(* CODESYS project systemdk.library
   Company: Beckhoff - DK
   DefaultNamespace: Tc3_SystemDK
   Title: Tc3_SystemDK
   Placeholder: Tc3_SystemDK
   Author: HCP
   Version: 3.3.1.5

Project tree, tasks and I/O mapping:
  libraries: Tc2_EtherCAT, * (Beckhoff Automation GmbH); Tc2_IoFunctions, * (Beckhoff Automation GmbH); Tc2_Standard, * (Beckhoff Automation GmbH); Tc2_SUPS, * (Beckhoff Automation GmbH); Tc2_System, * (Beckhoff Automation GmbH); Tc2_Utilities, * (Beckhoff Automation GmbH); Tc3_Interfaces, * (Beckhoff Automation GmbH); Tc3_Module, * (Beckhoff Automation GmbH)
  BASIC/
    POUs/
      FBs/
        DUTs/
          data type ST_Basic
          data type ST_Basic_Status
        GVLs/
          global variables GVL_Basic
        ITFs/
          interface I_Basic: M_nError, M_nReset, P_bAuto, P_bError, P_bManual, P_bReady, P_bReset, P_nErrorID
        function block FB_Basic [ST]: M_nError, M_nReset, P_bAuto, P_bError, P_bManual, P_bReady, P_bReset, P_nErrorID
  SYSTEM/
    POUs/
      FBs/
        DUTs/
          data type ST_EtherCATStatusDK
          data type ST_NovRamDK
          data type ST_SystemDK
          data type ST_WritePersistentDataDK
        ITFs/
          interface I_EtherCATStatusDK: M_nEnable, P_bWireBroke, P_nCfgSlaveCount, P_nDevState, P_nSlaveCount
          interface I_NovRamDK: M_nEnable
          interface I_SystemDK: M_nCerHost, M_nEnable, P_bIs_ARM, P_bIs_CE_Device, P_bIs_x64, P_bIs_x86, P_nAdsPort, P_nCycleTime, P_stDeviceIdentificationEx
          interface I_WritePersistentDataDK: M_n1_Second_UPS, M_nEnable, M_nWrite, P_bBusy, P_bPowerFailDetect, P_eSUPS_Mode, P_nWriteCNT
        function block FB_EtherCATStatusDK [ST]: M_nEnable, P_bWireBroke, P_nCfgSlaveCount, P_nDevState, P_nSlaveCount
        function block FB_NovRamDK [ST]: M_nEnable, M_nRead, M_nWrite
        function block FB_SystemDK [ST]: M_nCerHost, M_nEnable, P_bIs_ARM, P_bIs_CE_Device, P_bIs_x64, P_bIs_x86, P_nAdsPort, P_nCycleTime, P_stDeviceIdentificationEx
        function block FB_WritePersistentDataDK [ST]: M_n1_Second_UPS, M_nEnable, M_nWrite, P_bBusy, P_bPowerFailDetect, P_eSUPS_Mode, P_nWriteCNT
  Version/
    global variables Global_Version
*)

// BASIC/POUs/FBs/DUTs/ST_Basic
TYPE ST_Basic :
STRUCT
	bAuto: BOOL;
	bManual: BOOL;
	bReady: BOOL;
	bReset: BOOL;
	bError: BOOL;
	nErrorID: UDINT;
	nStatus: UDINT;	
	arr_nStatus: ARRAY[1..20] OF UDINT;
END_STRUCT
END_TYPE

// BASIC/POUs/FBs/DUTs/ST_Basic_Status
TYPE ST_Basic_Status :
STRUCT
	nError: UDINT;
	nReset:UDINT;
END_STRUCT
END_TYPE

// SYSTEM/POUs/FBs/DUTs/ST_EtherCATStatusDK
TYPE ST_EtherCATStatusDK EXTENDS ST_Basic :
STRUCT
	nDevState: UINT;
	nSlaveCount: UINT;
	nCfgSlaveCount: UINT;
	
	bWireBroke: BOOL;
END_STRUCT
END_TYPE

// SYSTEM/POUs/FBs/DUTs/ST_NovRamDK
TYPE ST_NovRamDK EXTENDS ST_Basic :
STRUCT
	bEnable: BOOL;
END_STRUCT
END_TYPE

// SYSTEM/POUs/FBs/DUTs/ST_SystemDK
TYPE ST_SystemDK EXTENDS ST_Basic :
STRUCT
	bIs_CE_Device: BOOL;			// Is a CE Device
	bIs_ARM: BOOL;					// Is ARM runtime
	bIs_x86: BOOL;					// Is x86 runtime
	bIs_x64: BOOL;					// Is x64 runtime
	nAdsPort: UINT;					// Plc port nr
	nCycleTime: UDINT;				// Plc cycle time in 100nS
	bCerHost_Enable: BOOL;			// Enable CerHost
	bCerHost_Disable: BOOL;			// Disable CerHost
	stDeviceIdentificationEx: Tc2_Utilities.ST_DeviceIdentificationEx;
END_STRUCT
END_TYPE

// SYSTEM/POUs/FBs/DUTs/ST_WritePersistentDataDK
TYPE ST_WritePersistentDataDK EXTENDS ST_Basic :
STRUCT
	bWrite: BOOL;
	bBusy: BOOL;
	bPowerFailDetect: BOOL;
	nWriteCNT: UDINT;
END_STRUCT
END_TYPE

// BASIC/POUs/FBs/GVLs/GVL_Basic
VAR_GLOBAL CONSTANT
	cIDLE: UDINT:= 0;						//	0 = idle
	cCOUPLED: UDINT:= 1;					//	1 = coupled
	cSTARTING: UDINT:= 2;					//	2 = starting
	cRUNNING: UDINT:= 3;					//	3 = running
	cABORTED: UDINT:= 4;					//	4 = aborted
	cNO_HARDWARE_CONNECTED: UDINT:= 5;		// 	5 = no hardware connected
	
	cPOINTER_OR_INDEX_ERROR: UDINT:= 7;		//	7 = pointer or index error
	cMAPPING_ERROR: UDINT:= 8;				//	8 = mapping error
	cPARAMETER_ERROR: UDINT:= 9;			//	9 = parameter error
	cCOMPLETE: UDINT:= 10;					//	10 = complete
END_VAR

// Version/Global_Version
// This function has been automatically generated from the project information.
VAR_GLOBAL CONSTANT
	{attribute 'const_non_replaced'}
	{attribute 'linkalways'}
	stLibVersion_Tc3_SystemDK : ST_LibVersion := (iMajor := 3, iMinor := 3, iBuild := 1, iRevision := 5, sVersion := '3.3.1.5');
END_VAR

// BASIC/POUs/FBs/ITFs/I_Basic
INTERFACE I_Basic

//	The result of the method is an unsigned double integer
//	0 = idle 
//	1 = coupled
//	2 = starting
//	3 = running
//	4 = aborted
// 	5 = no hardware connected
//	7 = pointer or index error
//	8 = mapping error
//	9 = parameter error
//	10 = complete
//	Any other number = ErrorID
METHOD PUBLIC M_nError : UDINT
VAR_INPUT
	nErrorID: UDINT;
END_VAR
END_METHOD

//	The result of the method is an unsigned double integer
//	0 = idle 
//	1 = coupled
//	2 = starting
//	3 = running
//	4 = aborted
// 	5 = no hardware connected
//	7 = pointer or index error
//	8 = mapping error
//	9 = parameter error
//	10 = complete
//	Any other number = ErrorID
METHOD PUBLIC M_nReset : UDINT
VAR_INPUT
	bExecute: BOOL;
END_VAR
END_METHOD

PROPERTY PUBLIC P_bAuto : BOOL
GET
END_GET
SET
END_SET
END_PROPERTY

PROPERTY PUBLIC P_bError : BOOL
GET
END_GET
END_PROPERTY

PROPERTY PUBLIC P_bManual : BOOL
GET
END_GET
SET
END_SET
END_PROPERTY

PROPERTY PUBLIC P_bReady : BOOL
GET
END_GET
SET
END_SET
END_PROPERTY

PROPERTY PUBLIC P_bReset : BOOL
GET
END_GET
END_PROPERTY

PROPERTY PUBLIC P_nErrorID : UDINT
GET
END_GET
END_PROPERTY

END_INTERFACE

// BASIC/POUs/FBs/FB_Basic
//------------------------------------------------------------------------------------------
//                                                                                        	
//***************************** Beckhoff TwinCAT Examples **********************************
//                                                                                        	
//************************************* WARNING ********************************************
// This program is only an example. If it is used as a control program in any real        	
// application, Beckhoff is not responsible for any malfunction, loss or damage           	
// which could arise by using this program!                                               	
//                                                                                        	
//*************************************  Program Info. *************************************
//                                                                                        	
// PLC program name:       FB_Basic (FB)               	                           	
// Hardware platform:      TwinCat v3.1.4012				                          	
// Modified by:            Hans Chr. Pallesen 			                                  	
//                                                                                        	
// ======================================================================================== 
//         Version       Date                        Remarks                              	
// ======================================================================================== 
//         1.0           17 feb 2013                 First release of this example        	
//         1.1           05 aug 2013                 Next release of this example        	
//         1.2           10 dec 2013                 Next release of this example        	
//         1.3           12 mar 2014                 Next release of this example        	
//         1.4           28 mar 2014                 Next release of this example        	
//         1.5           02 jun 2014                 Next release of this example        	
// ======================================================================================== 
//                                                                                        	
//******************************* Aims OF this PLC PROGRAM *********************************
//                                                                                        	
// Basic FB  						 			                               	
//																	                      	
//                                                                                        	
//----------------------------------------------------------------------------------------- 
FUNCTION_BLOCK FB_Basic IMPLEMENTS I_Basic
VAR
	_iIdx: INT;		// Temporary variabel - Index pointer
	
//*************************
// Property variables
//*************************
	_bReset: BOOL;
	_bAuto: BOOL := TRUE;
	_bManual: BOOL;
	_bError: BOOL;
	_nErrorID: UDINT;
	_bReady: BOOL;
	
//*************************
// Methods variable
//*************************
	FB_Basic_M_nReset_nScanCNT: UINT;
	FB_Basic_M_nReset_fbR_TRIG: Tc2_Standard.R_TRIG;
END_VAR

//	The result of the method is an unsigned double integer
//	0 = idle 
//	1 = coupled
//	2 = starting
//	3 = running
//	4 = aborted
// 	5 = no hardware connected
//	7 = pointer or index error
//	8 = mapping error
//	9 = parameter error
//	10 = complete
//	Any other number = ErrorID
METHOD PUBLIC M_nError : UDINT
VAR_INPUT
	nErrorID: UDINT;
END_VAR
//**********************************
// Update error
//**********************************
IF NOT _bError THEN
	_nErrorID:= nErrorID;
	_bError:= TRUE;
END_IF

M_nError:= cCOMPLETE;
END_METHOD

//	The result of the method is an unsigned double integer
//	0 = idle 
//	1 = coupled
//	2 = starting
//	3 = running
//	4 = aborted
// 	5 = no hardware connected
//	7 = pointer or index error
//	8 = mapping error
//	9 = parameter error
//	10 = complete
//	Any other number = ErrorID
METHOD PUBLIC M_nReset : UDINT
VAR_INPUT
	bExecute: BOOL;
END_VAR
//**********************************
// Wait for execute
//**********************************
FB_Basic_M_nReset_fbR_TRIG(CLK:= bExecute);
IF FB_Basic_M_nReset_fbR_TRIG.Q THEN
	FB_Basic_M_nReset_nScanCNT:= 4;	
	_bReset:= TRUE;
ELSE
	// Delay
	IF FB_Basic_M_nReset_nScanCNT = 0 THEN
		_bReset:= FALSE;
	ELSE
		IF FB_Basic_M_nReset_nScanCNT <= 2 THEN
			_bError:= FALSE;
			_nErrorID:= 16#00;
		END_IF	
	END_IF

	// Scan counter
	IF FB_Basic_M_nReset_nScanCNT > 0 THEN
		FB_Basic_M_nReset_nScanCNT:= FB_Basic_M_nReset_nScanCNT -1;
	ELSE	
		FB_Basic_M_nReset_nScanCNT:= 0;
	END_IF

	// Return method state
	IF bExecute THEN
		IF FB_Basic_M_nReset_nScanCNT = 0 THEN
			M_nReset:= cCOMPLETE;
		ELSE
			M_nReset:= cRUNNING;
		END_IF
	ELSE	
		M_nReset:= cIDLE;
	END_IF	
END_IF
END_METHOD

PROPERTY PUBLIC P_bAuto : BOOL
GET
P_bAuto:= _bAuto;
END_GET
SET
_bAuto:= P_bAuto;
END_SET
END_PROPERTY

PROPERTY PUBLIC P_bError : BOOL
GET
P_bError:= _bError;
END_GET
END_PROPERTY

PROPERTY PUBLIC P_bManual : BOOL
GET
P_bManual:= _bManual;
END_GET
SET
_bManual:= P_bManual;
END_SET
END_PROPERTY

PROPERTY PUBLIC P_bReady : BOOL
GET
P_bReady:= _bReady;
END_GET
SET
PUBLIC 
VAR
END_VAR
_bReady:= P_bReady;
END_SET
END_PROPERTY

PROPERTY PUBLIC P_bReset : BOOL
GET
P_bReset:= _bReset;
END_GET
END_PROPERTY

PROPERTY PUBLIC P_nErrorID : UDINT
GET
P_nErrorID:= _nErrorID;
END_GET
END_PROPERTY

END_FUNCTION_BLOCK

// SYSTEM/POUs/FBs/ITFs/I_EtherCATStatusDK
INTERFACE I_EtherCATStatusDK EXTENDS I_Basic

//	The result of the method is an unsigned double integer
//	0 = idle 
//	1 = coupled
//	2 = starting
//	3 = running
//	4 = aborted
// 	5 = no hardware connected
//	7 = pointer or index error
//	8 = mapping error
//	9 = parameter error
//	10 = complete
//	Any other number = ErrorID
METHOD PUBLIC M_nEnable : UDINT
VAR_INPUT
	bExecute: BOOL;
END_VAR
END_METHOD

PROPERTY PUBLIC P_bWireBroke : BOOL
GET
END_GET
END_PROPERTY

PROPERTY PUBLIC P_nCfgSlaveCount : UINT
GET
END_GET
END_PROPERTY

PROPERTY PUBLIC P_nDevState : UINT
GET
END_GET
END_PROPERTY

PROPERTY PUBLIC P_nSlaveCount : UINT
GET
END_GET
END_PROPERTY

END_INTERFACE

// SYSTEM/POUs/FBs/ITFs/I_NovRamDK
INTERFACE I_NovRamDK EXTENDS I_Basic

//	The result of the method is an unsigned double integer
//	0 = idle 
//	1 = coupled
//	2 = starting
//	3 = running
//	4 = aborted
// 	5 = no hardware connected
//	7 = pointer or index error
//	8 = mapping error
//	9 = parameter error
//	10 = complete
//	Any other number = ErrorID
METHOD M_nEnable : UDINT
VAR_INPUT
	bExecute: BOOL;
	nDevId: UINT;
	nMB_Offset: UINT;
	nMB_Size: UINT;
END_VAR
END_METHOD

END_INTERFACE

// SYSTEM/POUs/FBs/ITFs/I_SystemDK
INTERFACE I_SystemDK EXTENDS I_Basic

//	The result of the method is an unsigned double integer
//	0 = idle 
//	1 = coupled
//	2 = starting
//	3 = running
//	4 = aborted
// 	5 = no hardware connected
//	7 = pointer or index error
//	8 = mapping error
//	9 = parameter error
//	10 = complete
//	Any other number = ErrorID
METHOD PUBLIC M_nCerHost : UDINT
VAR_INPUT
	bEnable: BOOL;
	bDisable: BOOL;
END_VAR
END_METHOD

//	The result of the method is an unsigned double integer
//	0 = idle 
//	1 = coupled
//	2 = starting
//	3 = running
//	4 = aborted
// 	5 = no hardware connected
//	7 = pointer or index error
//	8 = mapping error
//	9 = parameter error
//	10 = complete
//	Any other number = ErrorID
METHOD PUBLIC M_nEnable : UDINT
VAR_INPUT
END_VAR
END_METHOD

PROPERTY PUBLIC P_bIs_ARM : BOOL
GET
END_GET
END_PROPERTY

PROPERTY PUBLIC P_bIs_CE_Device : BOOL
GET
END_GET
END_PROPERTY

PROPERTY PUBLIC P_bIs_x64 : BOOL
GET
END_GET
END_PROPERTY

PROPERTY PUBLIC P_bIs_x86 : BOOL
GET
END_GET
END_PROPERTY

PROPERTY PUBLIC P_nAdsPort : UINT
GET
END_GET
END_PROPERTY

PROPERTY PUBLIC P_nCycleTime : UDINT
GET
END_GET
END_PROPERTY

PROPERTY PUBLIC P_stDeviceIdentificationEx : Tc2_Utilities.ST_DeviceIdentificationEx
GET
END_GET
END_PROPERTY

END_INTERFACE

// SYSTEM/POUs/FBs/ITFs/I_WritePersistentDataDK
INTERFACE I_WritePersistentDataDK EXTENDS I_Basic

//	The result of the method is an unsigned double integer
//	0 = idle 
//	1 = coupled
//	2 = starting
//	3 = running
//	4 = aborted
// 	5 = no hardware connected
//	7 = pointer or index error
//	8 = mapping error
//	9 = parameter error
//	10 = complete
//	Any other number = ErrorID
METHOD PUBLIC M_n1_Second_UPS : UDINT
VAR_INPUT
	bExecute: BOOL;
END_VAR
END_METHOD

//	The result of the method is an unsigned double integer
//	0 = idle 
//	1 = coupled
//	2 = starting
//	3 = running
//	4 = aborted
// 	5 = no hardware connected
//	7 = pointer or index error
//	8 = mapping error
//	9 = parameter error
//	10 = complete
//	Any other number = ErrorID
METHOD M_nEnable : UDINT
VAR_INPUT
	bExecute: BOOL;
	tLogTimePuls: TIME;
END_VAR
END_METHOD

//	The result of the method is an unsigned double integer
//	0 = idle 
//	1 = coupled
//	2 = starting
//	3 = running
//	4 = aborted
// 	5 = no hardware connected
//	7 = pointer or index error
//	8 = mapping error
//	9 = parameter error
//	10 = complete
//	Any other number = ErrorID
METHOD M_nWrite : UDINT
VAR_INPUT
	bExecute: BOOL;
END_VAR
END_METHOD

PROPERTY PUBLIC P_bBusy : BOOL
GET
END_GET
END_PROPERTY

PROPERTY PUBLIC P_bPowerFailDetect : BOOL
GET
END_GET
END_PROPERTY

PROPERTY PUBLIC P_eSUPS_Mode : Tc2_SUPS.E_S_UPS_Mode
SET
END_SET
END_PROPERTY

PROPERTY PUBLIC P_nWriteCNT : UDINT
GET
END_GET
END_PROPERTY

END_INTERFACE

// SYSTEM/POUs/FBs/FB_EtherCATStatusDK
//------------------------------------------------------------------------------------------
//                                                                                        	
//***************************** Beckhoff TwinCAT Examples **********************************
//                                                                                        	
//************************************* WARNING ********************************************
// This program is only an example. If it is used as a control program in any real        	
// application, Beckhoff is not responsible for any malfunction, loss or damage           	
// which could arise by using this program!                                               	
//                                                                                        	
//*************************************  Program Info. *************************************
//                                                                                        	
// PLC program name:       FB_EtherCAT_Ok (FB)                                          	
// Hardware platform:      TwinCat v3.1.4014				                          	
// Modified by:            Hans Chr. Pallesen 			                                  	
//                                                                                        	
// ======================================================================================== 
//         Version       Date                        Remarks                              	
// ======================================================================================== 
//         1.0           12 feb 2014                 First release of this example        	
// ======================================================================================== 
//                                                                                        	
//******************************* Aims OF this PLC PROGRAM *********************************
//                                                                                        	
// Check EtherCAT state				 			                                      	
//																	                      	
//                                                                                        	
//----------------------------------------------------------------------------------------- 
FUNCTION_BLOCK FB_EtherCATStatusDK EXTENDS FB_Basic IMPLEMENTS I_EtherCATStatusDK
VAR
//**************************
// Static variables
//**************************
	AI_DevState AT %I*: UINT;
	AI_SlaveCount AT %I*: UINT;
	AI_CfgSlaveCount AT %I*: UINT;
//**************************
// Property variables
//**************************
	_bWireBroke: BOOL;
	
//**********************************
// Methods variable
//**********************************
	FB_EtherCATStatus_M_nEnable_fbDelay_TON: Tc2_Standard.TON;
END_VAR

//	The result of the method is an unsigned double integer
//	0 = idle 
//	1 = coupled
//	2 = starting
//	3 = running
//	4 = aborted
// 	5 = no hardware connected
//	7 = pointer or index error
//	8 = mapping error
//	9 = parameter error
//	10 = complete
//	Any other number = ErrorID
METHOD PUBLIC M_nEnable : UDINT
VAR_INPUT
	bExecute: BOOL;
END_VAR
// EtherCAT not configered
IF AI_SlaveCount = 0 AND AI_CfgSlaveCount = 0 THEN
	_bReady:= FALSE;
	_bWireBroke:= FALSE;
	M_nEnable:= cNO_HARDWARE_CONNECTED; 
ELSE
	// EtherCAT used
	IF bExecute THEN
		
		// Update Wire broke
		IF (AI_SlaveCount = 0 OR AI_SlaveCount <> AI_CfgSlaveCount) THEN
			M_nError(nErrorID:= 0);	
			_bWireBroke:= TRUE;
		ELSE
			_bWireBroke:= FALSE;
		END_IF
		
		// Update DevState
		IF AI_DevState <> 0 THEN
			M_nError(nErrorID:= 0);	
		END_IF
		
		// Method return value
		FB_EtherCATStatus_M_nEnable_fbDelay_TON(IN:= NOT _bWireBroke AND (AI_DevState = 0), PT:= T#100MS);
		_bReady:= FB_EtherCATStatus_M_nEnable_fbDelay_TON.Q;
		
		// Check for hardware
		IF AI_SlaveCount = 0 THEN
			M_nEnable:= cNO_HARDWARE_CONNECTED;
		ELSE
			IF _bReady THEN
				M_nEnable:= cCOMPLETE;
			ELSE
				M_nEnable:= cIDLE;
			END_IF
		END_IF
		
	ELSE
		FB_EtherCATStatus_M_nEnable_fbDelay_TON(IN:= FALSE);
		_bReady:= FALSE;
		_bWireBroke:= FALSE;
		M_nEnable:= cIDLE; 
	END_IF	

END_IF
END_METHOD

PROPERTY PUBLIC P_bWireBroke : BOOL
GET
P_bWireBroke:= _bWireBroke;
END_GET
END_PROPERTY

PROPERTY PUBLIC P_nCfgSlaveCount : UINT
GET
P_nCfgSlaveCount:= AI_CfgSlaveCount;
END_GET
END_PROPERTY

PROPERTY PUBLIC P_nDevState : UINT
GET
P_nDevState:= AI_DevState;
END_GET
END_PROPERTY

PROPERTY PUBLIC P_nSlaveCount : UINT
GET
P_nSlaveCount:= AI_SlaveCount;
END_GET
END_PROPERTY

END_FUNCTION_BLOCK

// SYSTEM/POUs/FBs/FB_NovRamDK
//------------------------------------------------------------------------------------------
//                                                                                        	
//***************************** Beckhoff TwinCAT Examples **********************************
//                                                                                        	
//************************************* WARNING ********************************************
// This program is only an example. If it is used as a control program in any real        	
// application, Beckhoff is not responsible for any malfunction, loss or damage           	
// which could arise by using this program!                                               	
//                                                                                        	
//*************************************  Program Info. *************************************
//                                                                                        	
// PLC program name:       FB_NovRamDK (FB)               	                           	
// Hardware platform:      TwinCat v3.1.4012				                          	
// Modified by:            Hans Chr. Pallesen 			                                  	
//                                                                                        	
// ======================================================================================== 
//         Version       Date                        Remarks                              	
// ======================================================================================== 
//         1.0           27 nov 2013                 First release of this example        	
// ======================================================================================== 
//                                                                                        	
//******************************* Aims OF this PLC PROGRAM *********************************
//                                                                                        	
//	Read/Write to NovRam																	                      	
//                                                                                        	
//----------------------------------------------------------------------------------------- 
FUNCTION_BLOCK FB_NovRamDK EXTENDS FB_Basic IMPLEMENTS I_NovRamDK
VAR
//**********************************
// Static variables
//**********************************
	_bEnable: BOOL;
	_nDevId: UINT;
	_nMB_Offset: UINT;
	_nMB_Size: UINT;
//**********************************
// Methods variable
//**********************************
	FB_NovRamDK_M_nEnable_nMBSrc AT %MB0: BYTE;
	FB_NovRamDK_M_nEnable_nBank: BYTE;
	FB_NovRamDK_M_nEnable_nCalcSize: UINT;
	FB_NovRamDK_M_nEnable_iState: UINT;
	FB_NovRamDK_M_nEnable_fbExecute_R_TRIG: Tc2_Standard.R_TRIG;
	FB_NovRamDK_M_nEnable_fbExecute_F_TRIG: Tc2_Standard.F_TRIG;
	FB_NovRamDK_M_nEnable_fbGetDPRAMInfo: Tc2_IoFunctions.FB_GetDPRAMInfo;
	FB_NovRamDK_M_nEnable_stNovRamAddrInfo: Tc2_IoFunctions.ST_NovRamAddrInfo;
	FB_NovRamDK_M_nEnable_nArrStatus: ARRAY[1..5] OF UDINT;

	FB_NovRamDK_M_nRead_fbNovRamReadWriteEx: FB_NovRamReadWriteEx;
	FB_NovRamDK_M_nRead_iState: UINT;
	FB_NovRamDK_M_nRead_nBank: BYTE;

	FB_NovRamDK_M_nWrite_fbNovRamReadWriteEx: FB_NovRamReadWriteEx;
	FB_NovRamDK_M_nWrite_bReady: BOOL;
	FB_NovRamDK_M_nWrite_iState: UINT;
	FB_NovRamDK_M_nWrite_nBank: BYTE;
	FB_NovRamDK_M_nWrite_pByte: POINTER TO BYTE;
	FB_NovRamDK_M_nWrite_pCard: POINTER TO BYTE;
END_VAR

//	The result of the method is an unsigned double integer
//	0 = idle 
//	1 = coupled
//	2 = starting
//	3 = running
//	4 = aborted
// 	5 = no hardware connected
//	7 = pointer or index error
//	8 = mapping error
//	9 = parameter error
//	10 = complete
//	Any other number = ErrorID
METHOD PUBLIC M_nEnable : UDINT
VAR_INPUT
	bExecute: BOOL;
	nDevId: UINT;
	nMB_Offset: UINT;
	nMB_Size: UINT;
END_VAR
//**********************************
// Local variable
//**********************************
THIS^._bEnable:= bExecute;
THIS^._nDevId:= nDevId;
THIS^._nMB_Offset:= nMB_Offset;
THIS^._nMB_Size:= nMB_Size;

//**********************************
// Reset
//**********************************
IF _bReset THEN
	IF _bError THEN
		FB_NovRamDK_M_nEnable_iState:= 000;
	END_IF
	M_nReset(bExecute:= _bReset);
END_IF

//**********************************
// Wait for execute
//**********************************
FB_NovRamDK_M_nEnable_fbExecute_R_TRIG(CLK:= bExecute);
FB_NovRamDK_M_nEnable_fbExecute_F_TRIG(CLK:= bExecute);
IF FB_NovRamDK_M_nEnable_fbExecute_R_TRIG.Q OR FB_NovRamDK_M_nEnable_fbExecute_F_TRIG.Q THEN
	FB_NovRamDK_M_nEnable_iState:= 000;
END_IF


//**********************************
// State maschine
//**********************************
CASE FB_NovRamDK_M_nEnable_iState OF
	
	000:	// Init
			_bReady:= FALSE; 
			FB_NovRamDK_M_nEnable_fbGetDPRAMInfo(bExecute:= FALSE); 
			IF M_nRead(bExecute:= FALSE) = cIDLE AND M_nWrite(bExecute:= FALSE) = cIDLE THEN
				FB_NovRamDK_M_nEnable_iState:= FB_NovRamDK_M_nEnable_iState +1;
			END_IF
	
	001:	// Wait for execute 
			IF bExecute THEN
				FB_NovRamDK_M_nEnable_iState:= FB_NovRamDK_M_nEnable_iState +1;
			END_IF
		
	002:	// Check parameter	
			M_nEnable:= cRUNNING;	
			IF _nDevId > 0 AND (nMB_Offset MOD 4 = 0) AND _nMB_Size > 0 AND (_nMB_Size MOD 4 = 0) THEN
				FB_NovRamDK_M_nEnable_iState:= FB_NovRamDK_M_nEnable_iState +1;
			ELSE
				M_nEnable:= cPARAMETER_ERROR;	
			END_IF	
		
	003:	// Calculate NovRam Size for ARM cpu
			M_nEnable:= cRUNNING;	
			IF (_nMB_Size + nMB_Offset) MOD 4 = 0 THEN
				FB_NovRamDK_M_nEnable_nCalcSize:= (_nMB_Size + nMB_Offset);
			ELSE
				FB_NovRamDK_M_nEnable_nCalcSize:= ((_nMB_Size + nMB_Offset) - (_nMB_Size + nMB_Offset MOD 4))+ 4;
			END_IF
			FB_NovRamDK_M_nEnable_iState:= FB_NovRamDK_M_nEnable_iState +1;
		
	004:	// Read NovRam size 
			M_nEnable:= cRUNNING;	
			FB_NovRamDK_M_nEnable_fbGetDPRAMInfo(
				nDevId:= _nDevId, 
				bExecute:= TRUE, 
				tTimeOut:= Tc2_System.DEFAULT_ADS_TIMEOUT, 
				bBusy=> , 
				bError=> , 
				nErrid=> , 
				stInfo=> FB_NovRamDK_M_nEnable_stNovRamAddrInfo);
	
			// Error
			IF FB_NovRamDK_M_nEnable_fbGetDPRAMInfo.bError THEN
				M_nError(nErrorID:= FB_NovRamDK_M_nEnable_fbGetDPRAMInfo.nErrId);
				M_nEnable:= FB_NovRamDK_M_nEnable_fbGetDPRAMInfo.nErrId;
			ELSE
				// Done
				IF NOT FB_NovRamDK_M_nEnable_fbGetDPRAMInfo.bBusy THEN
					FB_NovRamDK_M_nEnable_fbGetDPRAMInfo(bExecute:= FALSE); 
					FB_NovRamDK_M_nEnable_iState:= FB_NovRamDK_M_nEnable_iState +1;
				END_IF
			END_IF	
		
	005:	// Check max NovRam size
			M_nEnable:= cRUNNING;	
			IF FB_NovRamDK_M_nEnable_nCalcSize > ((FB_NovRamDK_M_nEnable_stNovRamAddrInfo.iCardMemSize/2) - 2) THEN
				FB_NovRamDK_M_nEnable_nCalcSize:= UDINT_TO_UINT(FB_NovRamDK_M_nEnable_stNovRamAddrInfo.iCardMemSize/2);
				FB_NovRamDK_M_nEnable_nCalcSize:= FB_NovRamDK_M_nEnable_nCalcSize - 4;
			END_IF
			FB_NovRamDK_M_nEnable_iState:= FB_NovRamDK_M_nEnable_iState +1;
	
	006:	// Read
			M_nEnable:= cRUNNING;	
			FB_NovRamDK_M_nEnable_nArrStatus[1]:= M_nRead(bExecute:= TRUE);
	
			// Error
			IF FB_NovRamDK_M_nEnable_nArrStatus[1] > cCOMPLETE THEN
				M_nError(nErrorID:= FB_NovRamDK_M_nEnable_nArrStatus[1]);
				M_nEnable:= FB_NovRamDK_M_nEnable_nArrStatus[1];
			ELSE
				// Done
				IF FB_NovRamDK_M_nEnable_nArrStatus[1] = cCOMPLETE THEN
					M_nRead(bExecute:= FALSE);
					FB_NovRamDK_M_nEnable_iState:= FB_NovRamDK_M_nEnable_iState +1;
				END_IF
			END_IF
			
	007:	// Write
			M_nEnable:= cRUNNING;	
			FB_NovRamDK_M_nEnable_nArrStatus[2]:= M_nWrite(bExecute:= TRUE);
			
			// Error
			IF FB_NovRamDK_M_nEnable_nArrStatus[2] > cCOMPLETE THEN
				M_nError(nErrorID:= FB_NovRamDK_M_nEnable_nArrStatus[2]);
				M_nEnable:= FB_NovRamDK_M_nEnable_nArrStatus[2];
			ELSE
				// Done
				IF FB_NovRamDK_M_nEnable_nArrStatus[2] = cCOMPLETE THEN
					M_nWrite(bExecute:= FALSE);
					FB_NovRamDK_M_nEnable_iState:= FB_NovRamDK_M_nEnable_iState +1;
				END_IF
			END_IF
	
	008:	// Done
			M_nEnable:= cCOMPLETE;	
			M_nWrite(bExecute:= TRUE);
			_bReady:= TRUE; 

ELSE
	FB_NovRamDK_M_nEnable_iState:= 000;
END_CASE
END_METHOD

//	The result of the method is an unsigned double integer
//	0 = idle 
//	1 = coupled
//	2 = starting
//	3 = running
//	4 = aborted
// 	5 = no hardware connected
//	7 = pointer or index error
//	8 = mapping error
//	9 = parameter error
//	10 = complete
//	Any other number = ErrorID
METHOD PRIVATE M_nRead : UDINT
VAR_INPUT
	bExecute: BOOL;
END_VAR
//**********************************
// Reset
//**********************************
IF _bReset THEN
	IF _bError THEN
		FB_NovRamDK_M_nRead_iState:= 000;
	END_IF
END_IF


//**********************************
// State maschine 
//**********************************
CASE FB_NovRamDK_M_nRead_iState OF

	000: 	// Init 
			FB_NovRamDK_M_nRead_fbNovRamReadWriteEx(bRead:= FALSE, bWrite:= FALSE);
			FB_NovRamDK_M_nRead_iState:= FB_NovRamDK_M_nRead_iState +1;

	001:	// Wait for execute 
			IF bExecute THEN
				FB_NovRamDK_M_nRead_iState:= FB_NovRamDK_M_nRead_iState +1;
			END_IF

	002:	// Read databank value 
			M_nRead:= cRUNNING;
			FB_NovRamDK_M_nRead_fbNovRamReadWriteEx(
				nDevId:= _nDevId,
				bRead:= TRUE,
				bWrite:= FALSE,
				cbSrcLen:= 1,
				cbDestLen:= 1,
				pSrcAddr:= ADR(FB_NovRamDK_M_nRead_nBank),
				pDestAddr:= ADR(FB_NovRamDK_M_nRead_nBank),
				nReadOffs:= FB_NovRamDK_M_nEnable_stNovRamAddrInfo.iCardMemSize -1,
				nWriteOffs:= 0,
				tTimeOut:= T#2s,
				_bBusy=> ,
				bError=> ,
				nErrId=> ,
				cbRead=> ,
				cbWrite=> );
	
			// Error	
			IF FB_NovRamDK_M_nRead_fbNovRamReadWriteEx.bError THEN
				M_nError(nErrorID:= FB_NovRamDK_M_nRead_fbNovRamReadWriteEx.nErrId);
				M_nRead:= FB_NovRamDK_M_nRead_fbNovRamReadWriteEx.nErrId;
			ELSE
				// Done
				IF NOT FB_NovRamDK_M_nRead_fbNovRamReadWriteEx.bBusy AND FB_NovRamDK_M_nRead_fbNovRamReadWriteEx.cbRead = 1 THEN
					FB_NovRamDK_M_nRead_fbNovRamReadWriteEx(bRead:= FALSE,	bWrite:= FALSE);
					FB_NovRamDK_M_nRead_iState:= FB_NovRamDK_M_nRead_iState +1;
				END_IF
			END_IF
	
	003:	// ReadNovRam data from databank 0 or 1 
			M_nRead:= cRUNNING;
			IF FB_NovRamDK_M_nRead_nBank = 0 THEN
				FB_NovRamDK_M_nRead_fbNovRamReadWriteEx(
					nDevId:= _nDevId,
					bRead:= TRUE,
					bWrite:= FALSE,
					cbSrcLen:= FB_NovRamDK_M_nEnable_nCalcSize,
					cbDestLen:= FB_NovRamDK_M_nEnable_nCalcSize,
					pSrcAddr:= ADR(FB_NovRamDK_M_nEnable_nMBSrc),
					pDestAddr:= ADR(FB_NovRamDK_M_nEnable_nMBSrc),
					nReadOffs:= 0,
					nWriteOffs:= 0,
					tTimeOut:= T#2s,
					_bBusy=> ,
					bError=> ,
					nErrId=> ,
					cbRead=> ,
					cbWrite=> );
			ELSE
				FB_NovRamDK_M_nRead_fbNovRamReadWriteEx(
					nDevId:= _nDevId,
					bRead:= TRUE,
					bWrite:= FALSE,
					cbSrcLen:= FB_NovRamDK_M_nEnable_nCalcSize,
					cbDestLen:= FB_NovRamDK_M_nEnable_nCalcSize,
					pSrcAddr:= ADR(FB_NovRamDK_M_nEnable_nMBSrc),
					pDestAddr:= ADR(FB_NovRamDK_M_nEnable_nMBSrc),
					nReadOffs:= FB_NovRamDK_M_nEnable_stNovRamAddrInfo.iCardMemSize / 2,
					nWriteOffs:= 0,
					tTimeOut:= T#2s,
					_bBusy=> ,
					bError=> ,
					nErrId=> ,
					cbRead=> ,
					cbWrite=> );
			END_IF
	
			// Error	
			IF FB_NovRamDK_M_nRead_fbNovRamReadWriteEx.bError THEN
				M_nError(nErrorID:= FB_NovRamDK_M_nRead_fbNovRamReadWriteEx.nErrId);
				M_nRead:= FB_NovRamDK_M_nRead_fbNovRamReadWriteEx.nErrId;
			ELSE
				// Done
				IF NOT FB_NovRamDK_M_nRead_fbNovRamReadWriteEx.bBusy AND FB_NovRamDK_M_nRead_fbNovRamReadWriteEx.cbRead = FB_NovRamDK_M_nEnable_nCalcSize THEN
					FB_NovRamDK_M_nRead_fbNovRamReadWriteEx(bRead:= FALSE,	bWrite:= FALSE);
					FB_NovRamDK_M_nRead_iState:= FB_NovRamDK_M_nRead_iState +1;
				END_IF
			END_IF
	
	004:	// Read done 
			M_nRead:= cCOMPLETE;
			IF NOT bExecute THEN
				FB_NovRamDK_M_nRead_iState:= 000;
			END_IF

ELSE
	FB_NovRamDK_M_nRead_iState:= 000;
END_CASE
END_METHOD

//	The result of the method is an unsigned double integer
//	0 = idle 
//	1 = coupled
//	2 = starting
//	3 = running
//	4 = aborted
// 	5 = no hardware connected
//	7 = pointer or index error
//	8 = mapping error
//	9 = parameter error
//	10 = complete
//	Any other number = ErrorID
METHOD PRIVATE M_nWrite : UDINT
VAR_INPUT
	bExecute: BOOL;
END_VAR
//**********************************
// Reset
//**********************************
IF _bReset THEN
	IF _bError THEN
		FB_NovRamDK_M_nWrite_iState:= 000;
	END_IF
END_IF


//**********************************
// State maschine 
//**********************************
CASE FB_NovRamDK_M_nWrite_iState OF

	000:	// Init
			FB_NovRamDK_M_nWrite_fbNovRamReadWriteEx(bRead:= FALSE,	bWrite:= FALSE);
			FB_NovRamDK_M_nWrite_bReady:= FALSE;
			FB_NovRamDK_M_nWrite_iState:= FB_NovRamDK_M_nWrite_iState +1;

	001:	// Wait for execute 
			IF bExecute THEN
				FB_NovRamDK_M_nWrite_iState:= FB_NovRamDK_M_nWrite_iState +1;
			END_IF

	002:	// Read databank value 
			M_nWrite:= cSTARTING;
			FB_NovRamDK_M_nWrite_fbNovRamReadWriteEx(
				nDevId:= _nDevId,
				bRead:= TRUE,
				bWrite:= FALSE,
				cbSrcLen:= 1,
				cbDestLen:= 1,
				pSrcAddr:= ADR(FB_NovRamDK_M_nWrite_nBank),
				pDestAddr:= ADR(FB_NovRamDK_M_nWrite_nBank),
				nReadOffs:= FB_NovRamDK_M_nEnable_stNovRamAddrInfo.iCardMemSize -1,
				nWriteOffs:= 0,
				tTimeOut:= T#2s,
				_bBusy=> ,
				bError=> ,
				nErrId=> ,
				cbRead=> ,
				cbWrite=> );
	
			// Error
			IF FB_NovRamDK_M_nWrite_fbNovRamReadWriteEx.bError THEN
				M_nError(nErrorID:= FB_NovRamDK_M_nWrite_fbNovRamReadWriteEx.nErrId);
				M_nWrite:= FB_NovRamDK_M_nWrite_fbNovRamReadWriteEx.nErrId;
			ELSE	
				// Done				
				IF FB_NovRamDK_M_nWrite_fbNovRamReadWriteEx.cbRead = 1 THEN
					FB_NovRamDK_M_nWrite_fbNovRamReadWriteEx(bRead:= FALSE,	bWrite:= FALSE);
					FB_NovRamDK_M_nWrite_iState:= FB_NovRamDK_M_nWrite_iState +1;
				END_IF
			END_IF
		
	003:	// Pointer settings 
			M_nWrite:= cSTARTING;
			FB_NovRamDK_M_nWrite_pByte:= ADR(FB_NovRamDK_M_nWrite_nBank);
			FB_NovRamDK_M_nWrite_pCard:= FB_NovRamDK_M_nEnable_stNovRamAddrInfo.pCardAddress + FB_NovRamDK_M_nEnable_stNovRamAddrInfo.iCardMemSize -1;
			FB_NovRamDK_M_nWrite_iState:= FB_NovRamDK_M_nWrite_iState +1;
		
	004:	// Write ready 
			M_nWrite:= cCOMPLETE;
			FB_NovRamDK_M_nWrite_bReady:= TRUE;
			IF NOT bExecute THEN
				FB_NovRamDK_M_nWrite_iState:= 000;
			END_IF
		
ELSE
	FB_NovRamDK_M_nWrite_iState:= 000;
END_CASE


// Write data to databank 0 or 1 
IF bExecute AND FB_NovRamDK_M_nWrite_bReady THEN
	IF FB_NovRamDK_M_nWrite_nBank = 1 THEN
		FB_NovRamDK_M_nWrite_nBank:= 0;
		MEMCPY(destAddr:= FB_NovRamDK_M_nEnable_stNovRamAddrInfo.pCardAddress, srcAddr:= ADR(FB_NovRamDK_M_nEnable_nMBSrc) + _nMB_Offset, n:= FB_NovRamDK_M_nEnable_nCalcSize);
		FB_NovRamDK_M_nWrite_pCard^:= FB_NovRamDK_M_nWrite_pByte^;
	ELSE
		FB_NovRamDK_M_nWrite_nBank:= 1;
		MEMCPY(destAddr:= FB_NovRamDK_M_nEnable_stNovRamAddrInfo.pCardAddress + (FB_NovRamDK_M_nEnable_stNovRamAddrInfo.iCardMemSize/2), srcAddr:= ADR(FB_NovRamDK_M_nEnable_nMBSrc) + _nMB_Offset, n:= FB_NovRamDK_M_nEnable_nCalcSize);
		FB_NovRamDK_M_nWrite_pCard^:= FB_NovRamDK_M_nWrite_pByte^;
	END_IF
END_IF
END_METHOD

END_FUNCTION_BLOCK

// SYSTEM/POUs/FBs/FB_SystemDK
//------------------------------------------------------------------------------------------
//                                                                                        	
//***************************** Beckhoff TwinCAT Examples **********************************
//                                                                                        	
//************************************* WARNING ********************************************
// This program is only an example. If it is used as a control program in any real        	
// application, Beckhoff is not responsible for any malfunction, loss or damage           	
// which could arise by using this program!                                               	
//                                                                                        	
//*************************************  Program Info. *************************************
//                                                                                        	
// PLC program name:       FB_SystemDK (FB)               	                           	
// Hardware platform:      TwinCat v3.1.4016				                          	
// Modified by:            Hans Chr. Pallesen 			                                  	
//                                                                                        	
// ======================================================================================== 
//         Version       Date                        Remarks                              	
// ======================================================================================== 
//         1.0           14 okt 2014                 First release of this example        	
// ======================================================================================== 
//                                                                                        	
//******************************* Aims OF this PLC PROGRAM *********************************
//                                                                                        	
//	TwinCAT device info																	                      	
//                                                                                        	
//----------------------------------------------------------------------------------------- 
FUNCTION_BLOCK FB_SystemDK EXTENDS FB_Basic IMPLEMENTS I_SystemDK
VAR
{attribute 'hide'}
	pInternPointer: POINTER TO INT;
END_VAR
VAR
//**************************
// Property variables
//**************************
	_bIs_ARM: BOOL;
	_stDeviceIdentificationEx: Tc2_Utilities.ST_DeviceIdentificationEx;

	
//**********************************
// Methods variable
//**********************************
	FB_SystemDK_M_nEnable_iState: INT;
	FB_SystemDK_M_nEnable_bDone: BOOL;
	FB_SystemDK_M_nEnable_stDeviceIdentificationEx: Tc2_Utilities.ST_DeviceIdentificationEx;
	FB_SystemDK_M_nEnable_fb_GetDeviceIdentificationEx: Tc2_Utilities.FB_GetDeviceIdentificationEx;
	
	FB_SystemDK_M_nCerHost_iState: INT;
	FB_SystemDK_M_nCerHost_sValue: STRING;
	FB_SystemDK_M_nCerHost_fbEnable_R_TRIG: Tc2_Standard.R_TRIG;
	FB_SystemDK_M_nCerHost_fbDisable_R_TRIG: Tc2_Standard.R_TRIG;
	FB_SystemDK_M_nCerHost_fbRegSetValue: Tc2_Utilities.FB_RegSetValue;
	FB_SystemDK_M_nCerHost_fbNT_Reboot: Tc2_Utilities.NT_Reboot;
END_VAR

//	The result of the method is an unsigned double integer
//	0 = idle 
//	1 = coupled
//	2 = starting
//	3 = running
//	4 = aborted
// 	5 = no hardware connected
//	7 = pointer or index error
//	8 = mapping error
//	9 = parameter error
//	10 = complete
//	Any other number = ErrorID
METHOD PUBLIC M_nCerHost : UDINT
VAR_INPUT
	bEnable: BOOL;
	bDisable: BOOL;
END_VAR
//**********************************
// Reset
//**********************************
IF _bReset THEN
	IF _bError THEN
		FB_SystemDK_M_nCerHost_fbRegSetValue(bExecute:= FALSE);
		FB_SystemDK_M_nCerHost_fbNT_Reboot(START:= FALSE); 
		FB_SystemDK_M_nCerHost_iState:= 000;
	END_IF
	M_nReset(bExecute:= _bReset);
END_IF

//**********************************
// Wait for execute
//**********************************
FB_SystemDK_M_nCerHost_fbEnable_R_TRIG(CLK:= bEnable);
IF FB_SystemDK_M_nCerHost_fbEnable_R_TRIG.Q THEN
	FB_SystemDK_M_nCerHost_fbRegSetValue(bExecute:= FALSE);
	FB_SystemDK_M_nCerHost_fbNT_Reboot(START:= FALSE); 
	FB_SystemDK_M_nCerHost_iState:= 001;
END_IF
FB_SystemDK_M_nCerHost_fbDisable_R_TRIG(CLK:= bDisable);
IF FB_SystemDK_M_nCerHost_fbDisable_R_TRIG.Q THEN
	FB_SystemDK_M_nCerHost_fbRegSetValue(bExecute:= FALSE);
	FB_SystemDK_M_nCerHost_fbNT_Reboot(START:= FALSE); 
	FB_SystemDK_M_nCerHost_iState:= 010;
END_IF


//**********************************
// State maschine
//**********************************
CASE FB_SystemDK_M_nCerHost_iState OF
	
	000:	// Do nothing
	
	001:	// Enable CerHost
			M_nCerHost:= cRUNNING;
			FB_SystemDK_M_nCerHost_sValue:= 'CeRDisp.exe';
			FB_SystemDK_M_nCerHost_fbRegSetValue(
				sNetId:= '', 
				sSubKey:= 'init', 
				sValName:= 'Launch90', 
				eValType:= REG_SZ, 
				cbData:= INT_TO_UDINT(Tc2_Standard.LEN(FB_SystemDK_M_nCerHost_sValue)), 
				pData:= ADR(FB_SystemDK_M_nCerHost_sValue), 
				bExecute:= TRUE, 
				tTimeOut:= Tc2_System.DEFAULT_ADS_TIMEOUT, 
				bBusy=> , 
				bError=> , 
				nErrId=> , 
				cbWrite=> );
		
			// Error	
			IF FB_SystemDK_M_nCerHost_fbRegSetValue.bError THEN
				M_nError(nErrorID:= FB_SystemDK_M_nCerHost_fbRegSetValue.nErrId);
				M_nCerHost:= FB_SystemDK_M_nCerHost_fbRegSetValue.nErrId;
			ELSE
				// Done
				IF NOT FB_SystemDK_M_nCerHost_fbRegSetValue.bBusy THEN
					FB_SystemDK_M_nCerHost_fbRegSetValue(bExecute:= FALSE);
					FB_SystemDK_M_nCerHost_iState:= FB_SystemDK_M_nCerHost_iState +1;
				END_IF
			END_IF
	
	002:	// Enable done
			M_nCerHost:= cRUNNING;
			FB_SystemDK_M_nCerHost_iState:= 20;

	010:	// Disable CerHost
			M_nCerHost:= cRUNNING;
			FB_SystemDK_M_nCerHost_sValue:= '_CeRDisp.exe';
			FB_SystemDK_M_nCerHost_fbRegSetValue(
				sNetId:= '', 
				sSubKey:= 'init', 
				sValName:= 'Launch90', 
				eValType:= REG_SZ, 
				cbData:= INT_TO_UDINT(Tc2_Standard.LEN(FB_SystemDK_M_nCerHost_sValue)), 
				pData:= ADR(FB_SystemDK_M_nCerHost_sValue), 
				bExecute:= TRUE, 
				tTimeOut:= Tc2_System.DEFAULT_ADS_TIMEOUT, 
				bBusy=> , 
				bError=> , 
				nErrId=> , 
				cbWrite=> );
		
			// Error	
			IF FB_SystemDK_M_nCerHost_fbRegSetValue.bError THEN
				M_nError(nErrorID:= FB_SystemDK_M_nCerHost_fbRegSetValue.nErrId);
				M_nCerHost:= FB_SystemDK_M_nCerHost_fbRegSetValue.nErrId;
			ELSE
				// Done
				IF NOT FB_SystemDK_M_nCerHost_fbRegSetValue.bBusy THEN
					FB_SystemDK_M_nCerHost_fbRegSetValue(bExecute:= FALSE);
					FB_SystemDK_M_nCerHost_iState:= FB_SystemDK_M_nCerHost_iState +1;
				END_IF
			END_IF
			
	011:	// Disable done
			M_nCerHost:= cRUNNING;
			FB_SystemDK_M_nCerHost_iState:= 20;

	020:	// Reboot
			M_nCerHost:= cRUNNING;
			FB_SystemDK_M_nCerHost_fbNT_Reboot(
				NETID:= '', 
				DELAY:= 0, 
				START:= TRUE, 
				TMOUT:= Tc2_System.DEFAULT_ADS_TIMEOUT, 
				BUSY=> , 
				ERR=> , 
				ERRID=> );
	
			// Error	
			IF FB_SystemDK_M_nCerHost_fbNT_Reboot.ERR THEN
				M_nError(nErrorID:= FB_SystemDK_M_nCerHost_fbNT_Reboot.ERRID);
				M_nCerHost:= FB_SystemDK_M_nCerHost_fbNT_Reboot.ERRID;
			END_IF
		
ELSE
	FB_SystemDK_M_nCerHost_iState:= 000;
END_CASE
END_METHOD

//	The result of the method is an unsigned double integer
//	0 = idle 
//	1 = coupled
//	2 = starting
//	3 = running
//	4 = aborted
// 	5 = no hardware connected
//	7 = pointer or index error
//	8 = mapping error
//	9 = parameter error
//	10 = complete
//	Any other number = ErrorID
METHOD PUBLIC M_nEnable : UDINT
VAR_INPUT
END_VAR
//**********************************
// Reset
//**********************************
IF _bReset THEN
	IF NOT FB_SystemDK_M_nEnable_bDone THEN
		FB_SystemDK_M_nEnable_fb_GetDeviceIdentificationEx(bExecute:= FALSE); 
		FB_SystemDK_M_nEnable_iState:= 000;
	END_IF
	M_nReset(bExecute:= _bReset);
END_IF

// Status
IF _stDeviceIdentificationEx.strHardwareCPU = 'ARM' THEN
	_bIs_ARM:= TRUE;
ELSE
	_bIs_ARM:= FALSE;
END_IF

//**********************************
// State maschine
//**********************************
CASE FB_SystemDK_M_nEnable_iState OF
	
	000:	// Init
			FB_SystemDK_M_nEnable_fb_GetDeviceIdentificationEx(bExecute:= FALSE); 
			FB_SystemDK_M_nEnable_bDone:= FALSE;
			FB_SystemDK_M_nEnable_iState:= FB_SystemDK_M_nEnable_iState +1;
		
	001:	// Get data	
			M_nEnable:= cRUNNING;
			FB_SystemDK_M_nEnable_fb_GetDeviceIdentificationEx(bExecute:= FALSE); 
			FB_SystemDK_M_nEnable_fb_GetDeviceIdentificationEx(
				bExecute:= TRUE, 
				tTimeout:= Tc2_System.DEFAULT_ADS_TIMEOUT, 
				sNetId:= '', 
				bBusy=> , 
				bError=> , 
				nErrorID=> , 
				stDevIdent=> FB_SystemDK_M_nEnable_stDeviceIdentificationEx);
	
			FB_SystemDK_M_nEnable_iState:= FB_SystemDK_M_nEnable_iState +1;
	
	002:	// Get data done
			M_nEnable:= cRUNNING;
			FB_SystemDK_M_nEnable_fb_GetDeviceIdentificationEx(bExecute:= TRUE, stDevIdent=> FB_SystemDK_M_nEnable_stDeviceIdentificationEx);
			IF FB_SystemDK_M_nEnable_fb_GetDeviceIdentificationEx.bError THEN
				M_nError(nErrorID:= FB_SystemDK_M_nEnable_fb_GetDeviceIdentificationEx.nErrorID);
				M_nEnable:= FB_SystemDK_M_nEnable_fb_GetDeviceIdentificationEx.nErrorID;
			ELSE
				// Done
				IF NOT FB_SystemDK_M_nEnable_fb_GetDeviceIdentificationEx.bBusy THEN
					_stDeviceIdentificationEx:= FB_SystemDK_M_nEnable_stDeviceIdentificationEx;
					FB_SystemDK_M_nEnable_fb_GetDeviceIdentificationEx(bExecute:= FALSE); 
					FB_SystemDK_M_nEnable_iState:= FB_SystemDK_M_nEnable_iState +1;
				END_IF	
			END_IF
		
	003:	// Done	
			M_nEnable:= cCOMPLETE;
			FB_SystemDK_M_nEnable_bDone:= TRUE;

ELSE
	FB_SystemDK_M_nEnable_iState:= 000;
END_CASE


// bReady
IF FB_SystemDK_M_nEnable_bDone THEN
	_bReady:= TRUE;
ELSE
	_bReady:= FALSE;
END_IF
END_METHOD

PROPERTY PUBLIC P_bIs_ARM : BOOL
GET
P_bIs_ARM:= _bIs_ARM;
END_GET
END_PROPERTY

PROPERTY PUBLIC P_bIs_CE_Device : BOOL
GET
P_bIs_CE_Device:= _stDeviceIdentificationEx.strImageOsName = 'Windows CE';
END_GET
END_PROPERTY

PROPERTY PUBLIC P_bIs_x64 : BOOL
GET
IF _bIs_ARM THEN
	P_bIs_x64:= FALSE;
ELSE
	IF SIZEOF(pInternPointer) > 4 THEN
		P_bIs_x64:= TRUE;
	ELSE
		P_bIs_x64:= FALSE;
	END_IF	
END_IF
END_GET
END_PROPERTY

PROPERTY PUBLIC P_bIs_x86 : BOOL
GET
IF _bIs_ARM THEN
	P_bIs_x86:= FALSE;
ELSE
	IF SIZEOF(pInternPointer) = 4 THEN
		P_bIs_x86:= TRUE;
	ELSE
		P_bIs_x86:= FALSE;
	END_IF	
END_IF
END_GET
END_PROPERTY

PROPERTY PUBLIC P_nAdsPort : UINT
GET
P_nAdsPort:= TwinCAT_SystemInfoVarList._AppInfo.AdsPort;
END_GET
END_PROPERTY

PROPERTY PUBLIC P_nCycleTime : UDINT
GET
P_nCycleTime:= TwinCAT_SystemInfoVarList._TaskInfo[Tc2_System.GETCURTASKINDEXEX()].CycleTime;
END_GET
END_PROPERTY

PROPERTY PUBLIC P_stDeviceIdentificationEx : Tc2_Utilities.ST_DeviceIdentificationEx
GET
P_stDeviceIdentificationEx:= _stDeviceIdentificationEx;
END_GET
END_PROPERTY

END_FUNCTION_BLOCK

// SYSTEM/POUs/FBs/FB_WritePersistentDataDK
//------------------------------------------------------------------------------------------
//                                                                                        	
//***************************** Beckhoff TwinCAT Examples **********************************
//                                                                                        	
//************************************* WARNING ********************************************
// This program is only an example. If it is used as a control program in any real        	
// application, Beckhoff is not responsible for any malfunction, loss or damage           	
// which could arise by using this program!                                               	
//                                                                                        	
//*************************************  Program Info. *************************************
//                                                                                        	
// PLC program name:       FB_WritePersistentDataDK (FB)                                          	
// Hardware platform:      TwinCat v3.1.4012				                          	
// Modified by:            Hans Chr. Pallesen 			                                  	
//                                                                                        	
// ======================================================================================== 
//         Version       Date                        Remarks                              	
// ======================================================================================== 
//         1.0           02 feb 2014                 First release of this example        	
// ======================================================================================== 
//                                                                                        	
//******************************* Aims OF this PLC PROGRAM *********************************
//                                                                                        	
// Write persistent data file				 			                                      	
//																	                      	
//                                                                                        	
//----------------------------------------------------------------------------------------- 
FUNCTION_BLOCK FB_WritePersistentDataDK EXTENDS FB_Basic IMPLEMENTS I_WritePersistentDataDK
VAR
//**************************
// Static variables
//**************************
	_bFirstBoot: BOOL := TRUE;
	_nAdsPort: UINT;
	_bPowerFailDetect: BOOL;
	_fbWritePersistentData: Tc2_Utilities.FB_WritePersistentData;
	_nWriteCNT: UDINT;
	_eUpsMode: Tc2_SUPS.E_S_UPS_Mode;
	
//**************************
// Property variables
//**************************
	_bBusy: BOOL;	
	
//**************************
// Methods variable
//**************************

	FB_WritePersistentDataDK_M_nEnable_iState: INT;
	FB_WritePersistentDataDK_M_nEnable_fbExecute_R_TRIG: R_TRIG;
	FB_WritePersistentDataDK_M_nEnable_fbReset_R_TRIG: R_TRIG;
	FB_WritePersistentDataDK_M_nEnable_fbStartDelay_TON: TON;
	FB_WritePersistentDataDK_M_nEnable_fbLogTimePuls_TON: TON;
	
	FB_WritePersistentDataDK_M_nWrite_iState: INT;
	FB_WritePersistentDataDK_M_nWrite_fbExecute_R_TRIG: R_TRIG;
	FB_WritePersistentDataDK_M_nWrite_fbReset_R_TRIG: R_TRIG;
	FB_WritePersistentDataDK_M_nWrite_fbStartDelay_TON: TON;
	
	FB_WritePersistentDataDK_M_n1_Second_UPS_iState: INT;
	FB_WritePersistentDataDK_M_n1_Second_UPS_bIs_CB3011: BOOL;
	FB_WritePersistentDataDK_M_n1_Second_UPS_bIs_CX9020_U900: BOOL;
	FB_WritePersistentDataDK_M_n1_Second_UPS_bIs_CX50x0: BOOL;
	FB_WritePersistentDataDK_M_n1_Second_UPS_bIs_CX51x0: BOOL;
	
	FB_WritePersistentDataDK_M_n1_Second_UPS_fb_S_UPS_CB3011: Tc2_SUPS.FB_S_UPS_CB3011; 
	FB_WritePersistentDataDK_M_n1_Second_UPS_fb_S_UPS_CX9020_U900: Tc2_SUPS.FB_S_UPS_CX9020_U900; 
	FB_WritePersistentDataDK_M_n1_Second_UPS_fb_S_UPS_CX50x0: Tc2_SUPS.FB_S_UPS;
	FB_WritePersistentDataDK_M_n1_Second_UPS_fb_S_UPS_CX51x0: Tc2_SUPS.FB_S_UPS_CX51x0;
	
	FB_WritePersistentDataDK_M_n1_Second_UPS_stDeviceIdentificationEx: Tc2_Utilities.ST_DeviceIdentificationEx;
	FB_WritePersistentDataDK_M_n1_Second_UPS_fb_GetDeviceIdentificationEx: Tc2_Utilities.FB_GetDeviceIdentificationEx;
	
END_VAR

//	The result of the method is an unsigned double integer
//	0 = idle 
//	1 = coupled
//	2 = starting
//	3 = running
//	4 = aborted
// 	5 = no hardware connected
//	7 = pointer or index error
//	8 = mapping error
//	9 = parameter error
//	10 = complete
//	Any other number = ErrorID
METHOD PUBLIC M_n1_Second_UPS : UDINT
VAR_INPUT
	bExecute: BOOL;
END_VAR
_bPowerFailDetect:= FALSE;

// Update CX9020-U900 UPS
IF FB_WritePersistentDataDK_M_n1_Second_UPS_bIs_CB3011 THEN
	
	FB_WritePersistentDataDK_M_n1_Second_UPS_fb_S_UPS_CB3011(
		sNetID:= , 
		iPLCPort:= TwinCAT_SystemInfoVarList._AppInfo.AdsPort, 
		tTimeout:= , 
		eUpsMode:= _eUpsMode, 
		ePersistentMode:= , 
		tRecoverTime:= , 
		bPowerFailDetect=> _bPowerFailDetect, 
		eState=> );

END_IF

// Update CX9020-U900 UPS
IF FB_WritePersistentDataDK_M_n1_Second_UPS_bIs_CX9020_U900 THEN

	FB_WritePersistentDataDK_M_n1_Second_UPS_fb_S_UPS_CX9020_U900(
		sNetID:= , 
		iPLCPort:= TwinCAT_SystemInfoVarList._AppInfo.AdsPort, 
		tTimeout:= , 
		eUpsMode:= _eUpsMode, 
		ePersistentMode:= , 
		tRecoverTime:= , 
		bPowerFailDetect=> _bPowerFailDetect, 
		eState=> );

END_IF

// Update CX50x0 UPS
IF FB_WritePersistentDataDK_M_n1_Second_UPS_bIs_CX50x0 THEN
	
	FB_WritePersistentDataDK_M_n1_Second_UPS_fb_S_UPS_CX50x0(
		sNetID:= , 
		iPLCPort:= TwinCAT_SystemInfoVarList._AppInfo.AdsPort, 
		iUPSPort:= , 
		tTimeout:= , 
		eUpsMode:= _eUpsMode, 
		ePersistentMode:= , 
		tRecoverTime:= , 
		bPowerFailDetect=> _bPowerFailDetect, 
		eState=> );

END_IF

// Update CX51x0 UPS
IF FB_WritePersistentDataDK_M_n1_Second_UPS_bIs_CX51x0 THEN
		
	FB_WritePersistentDataDK_M_n1_Second_UPS_fb_S_UPS_CX51x0(
		sNetID:= , 
		iPLCPort:= TwinCAT_SystemInfoVarList._AppInfo.AdsPort, 
		iUPSPort:= , 
		tTimeout:= , 
		eUpsMode:= _eUpsMode, 
		ePersistentMode:= , 
		tRecoverTime:= , 
		bPowerFailDetect=> _bPowerFailDetect, 
		eState=> );

END_IF

	
//**********************************
// Reset 
//**********************************
IF _bReset THEN
	IF _bError THEN	
		FB_WritePersistentDataDK_M_n1_Second_UPS_iState:= 000;
	END_IF	
END_IF


//**********************************
// State maschine
//**********************************
CASE FB_WritePersistentDataDK_M_n1_Second_UPS_iState OF
	
	000:	// Wait for execute and start delay
			IF bExecute THEN
				IF FB_WritePersistentDataDK_M_nEnable_fbStartDelay_TON.Q THEN
					FB_WritePersistentDataDK_M_n1_Second_UPS_iState:= FB_WritePersistentDataDK_M_n1_Second_UPS_iState +1;
				END_IF
			END_IF	

	001:	// Get data	
			M_n1_Second_UPS:= cRUNNING;
			FB_WritePersistentDataDK_M_n1_Second_UPS_fb_GetDeviceIdentificationEx(bExecute:= FALSE); 
			FB_WritePersistentDataDK_M_n1_Second_UPS_fb_GetDeviceIdentificationEx(
				bExecute:= TRUE, 
				tTimeout:= Tc2_System.DEFAULT_ADS_TIMEOUT, 
				sNetId:= '', 
				bBusy=> , 
				bError=> , 
				nErrorID=> , 
				stDevIdent=> FB_WritePersistentDataDK_M_n1_Second_UPS_stDeviceIdentificationEx);
	
			FB_WritePersistentDataDK_M_n1_Second_UPS_iState:= FB_WritePersistentDataDK_M_n1_Second_UPS_iState +1;
	
	002:	// Get data done
			M_n1_Second_UPS:= cRUNNING;
			FB_WritePersistentDataDK_M_n1_Second_UPS_fb_GetDeviceIdentificationEx(bExecute:= FALSE, stDevIdent=> FB_WritePersistentDataDK_M_n1_Second_UPS_stDeviceIdentificationEx);
			IF FB_WritePersistentDataDK_M_n1_Second_UPS_fb_GetDeviceIdentificationEx.bError THEN
				M_nError(nErrorID:= FB_WritePersistentDataDK_M_n1_Second_UPS_fb_GetDeviceIdentificationEx.nErrorID);
				M_n1_Second_UPS:= FB_WritePersistentDataDK_M_n1_Second_UPS_fb_GetDeviceIdentificationEx.nErrorID;
			ELSE
				// Done
				IF NOT FB_WritePersistentDataDK_M_n1_Second_UPS_fb_GetDeviceIdentificationEx.bBusy THEN
					FB_WritePersistentDataDK_M_n1_Second_UPS_iState:= FB_WritePersistentDataDK_M_n1_Second_UPS_iState +1;
				END_IF	
			END_IF
		
	003:	// Check 1s UPS device type
			M_n1_Second_UPS:= cRUNNING;
			FB_WritePersistentDataDK_M_n1_Second_UPS_bIs_CB3011:= Tc2_Standard.MID(FB_WritePersistentDataDK_M_n1_Second_UPS_stDeviceIdentificationEx.strHardwareModel, 5, 1) = 'CB3011';
			FB_WritePersistentDataDK_M_n1_Second_UPS_bIs_CX9020_U900:= Tc2_Standard.MID(FB_WritePersistentDataDK_M_n1_Second_UPS_stDeviceIdentificationEx.strHardwareModel, 11, 1) = 'CX9020-U900';
			FB_WritePersistentDataDK_M_n1_Second_UPS_bIs_CX50x0:= Tc2_Standard.MID(FB_WritePersistentDataDK_M_n1_Second_UPS_stDeviceIdentificationEx.strHardwareModel, 2, 1) = '50';
			FB_WritePersistentDataDK_M_n1_Second_UPS_bIs_CX51x0:= Tc2_Standard.MID(FB_WritePersistentDataDK_M_n1_Second_UPS_stDeviceIdentificationEx.strHardwareModel, 4, 1) = 'CX51';
		
			// 1s UPS hardware connected
			IF FB_WritePersistentDataDK_M_n1_Second_UPS_bIs_CB3011 THEN
				FB_WritePersistentDataDK_M_n1_Second_UPS_iState:= FB_WritePersistentDataDK_M_n1_Second_UPS_iState +2;
			ELSE
				IF FB_WritePersistentDataDK_M_n1_Second_UPS_bIs_CX9020_U900 THEN
					FB_WritePersistentDataDK_M_n1_Second_UPS_iState:= FB_WritePersistentDataDK_M_n1_Second_UPS_iState +2;
				ELSE
					IF FB_WritePersistentDataDK_M_n1_Second_UPS_bIs_CX50x0 THEN
						FB_WritePersistentDataDK_M_n1_Second_UPS_iState:= FB_WritePersistentDataDK_M_n1_Second_UPS_iState +2;
					ELSE
						IF FB_WritePersistentDataDK_M_n1_Second_UPS_bIs_CX51x0 THEN
							FB_WritePersistentDataDK_M_n1_Second_UPS_iState:= FB_WritePersistentDataDK_M_n1_Second_UPS_iState +2;
						ELSE
							FB_WritePersistentDataDK_M_n1_Second_UPS_iState:= FB_WritePersistentDataDK_M_n1_Second_UPS_iState +1;
						END_IF
					END_IF
				END_IF	
			END_IF

	004:	// No 1sec UPS hardware connected	
			IF bExecute THEN
				M_n1_Second_UPS:= cNO_HARDWARE_CONNECTED;
			ELSE
				FB_WritePersistentDataDK_M_n1_Second_UPS_iState:= 000;
			END_IF	

	005:	// Start delay
			M_n1_Second_UPS:= cRUNNING;
			IF bExecute THEN
				IF FB_WritePersistentDataDK_M_nEnable_fbStartDelay_TON.Q THEN
					FB_WritePersistentDataDK_M_n1_Second_UPS_iState:= FB_WritePersistentDataDK_M_n1_Second_UPS_iState +1;
				END_IF
			ELSE
				FB_WritePersistentDataDK_M_n1_Second_UPS_iState:= 000;
			END_IF	
	
	006:	// Wait not Execute
			M_n1_Second_UPS:= cCOMPLETE;
			IF NOT bExecute THEN
				FB_WritePersistentDataDK_M_n1_Second_UPS_iState:= 000;
			END_IF	

ELSE
	FB_WritePersistentDataDK_M_n1_Second_UPS_iState:= 000;
END_CASE
END_METHOD

//	The result of the method is an unsigned double integer
//	0 = idle 
//	1 = coupled
//	2 = starting
//	3 = running
//	4 = aborted
// 	5 = no hardware connected
//	7 = pointer or index error
//	8 = mapping error
//	9 = parameter error
//	10 = complete
//	Any other number = ErrorID
METHOD PUBLIC M_nEnable : UDINT
VAR_INPUT
	bExecute: BOOL;
	tLogTimePuls: TIME;
END_VAR
// Local variable
THIS^._nAdsPort:= TwinCAT_SystemInfoVarList._AppInfo.AdsPort;

//**********************************
// Reset 
//**********************************
IF _bReset THEN
	IF _bError THEN	
		FB_WritePersistentDataDK_M_nEnable_iState:= 000;
	END_IF	
	M_nReset(bExecute:= _bReset);
END_IF

// Power fail
FB_WritePersistentDataDK_M_nEnable_fbReset_R_TRIG(CLK:= _bPowerFailDetect, Q=> );
IF FB_WritePersistentDataDK_M_nEnable_fbReset_R_TRIG.Q THEN
	FB_WritePersistentDataDK_M_nEnable_iState:= 000;
END_IF

// Startup delay
FB_WritePersistentDataDK_M_nEnable_fbStartDelay_TON(IN:= TRUE, PT:= T#15S);

// LogTtime puls
IF FB_WritePersistentDataDK_M_nEnable_fbStartDelay_TON.Q THEN
	FB_WritePersistentDataDK_M_nEnable_fbLogTimePuls_TON(IN:= bExecute AND tLogTimePuls > T#0MS AND NOT FB_WritePersistentDataDK_M_nEnable_fbLogTimePuls_TON.Q, PT:= tLogTimePuls);
ELSE
	FB_WritePersistentDataDK_M_nEnable_fbLogTimePuls_TON(IN:= FALSE);
END_IF	

//**********************************
// Wait for execute
//**********************************
IF FB_WritePersistentDataDK_M_nEnable_fbStartDelay_TON.Q THEN
	FB_WritePersistentDataDK_M_nEnable_fbExecute_R_TRIG(CLK:= (_bFirstBoot OR FB_WritePersistentDataDK_M_nEnable_fbLogTimePuls_TON.Q) AND NOT _bPowerFailDetect);
	IF FB_WritePersistentDataDK_M_nEnable_fbExecute_R_TRIG.Q THEN
		FB_WritePersistentDataDK_M_nEnable_iState:= 001;
	END_IF
ELSE
	FB_WritePersistentDataDK_M_nEnable_fbExecute_R_TRIG(CLK:= FALSE);
	FB_WritePersistentDataDK_M_nEnable_iState:= 000;
END_IF


//**********************************
// Main sekvens
//**********************************
CASE FB_WritePersistentDataDK_M_nEnable_iState OF

	000:	// Do nothing
			IF _bError THEN
				M_nEnable:= _nErrorID;
			ELSE
				IF bExecute THEN
					IF FB_WritePersistentDataDK_M_nEnable_fbStartDelay_TON.Q THEN
						M_nEnable:= cCOMPLETE;
					ELSE
						M_nEnable:= cSTARTING;
					END_IF
				END_IF	
			END_IF

	001:	// Init
			M_nEnable:= cSTARTING;
			_fbWritePersistentData.PORT:= _nAdsPort;
			_fbWritePersistentData.TMOUT:= Tc2_System.DEFAULT_ADS_TIMEOUT;
			FB_WritePersistentDataDK_M_nEnable_iState:= FB_WritePersistentDataDK_M_nEnable_iState +1;

	002:	// Running
			M_nEnable:= cSTARTING;
			IF _fbWritePersistentData.BUSY THEN
				FB_WritePersistentDataDK_M_nEnable_iState:= FB_WritePersistentDataDK_M_nEnable_iState +3;
			ELSE
				FB_WritePersistentDataDK_M_nEnable_iState:= FB_WritePersistentDataDK_M_nEnable_iState +1;
			END_IF
			
	003:	// Init
			M_nEnable:= cSTARTING;
			_fbWritePersistentData.START:= FALSE; 
			FB_WritePersistentDataDK_M_nEnable_iState:= FB_WritePersistentDataDK_M_nEnable_iState +1;

	004:	// Start
			M_nEnable:= cSTARTING;
			_fbWritePersistentData.START:= TRUE; 
			FB_WritePersistentDataDK_M_nEnable_iState:= FB_WritePersistentDataDK_M_nEnable_iState +1;

	005:	// Write persistent data - Done
			M_nEnable:= cSTARTING;
		
			// Error handling
			IF _fbWritePersistentData.ERR THEN
				M_nError(nErrorID:= _fbWritePersistentData.ERRID);	
				M_nEnable:= _fbWritePersistentData.ERRID;
			ELSE
				// Done
				IF NOT _fbWritePersistentData.BUSY THEN
					IF _bFirstBoot THEN
						_fbWritePersistentData.START:= FALSE; 
						FB_WritePersistentDataDK_M_nEnable_iState:= FB_WritePersistentDataDK_M_nEnable_iState +1;
					ELSE
						_nWriteCNT:= _nWriteCNT +1;
						_fbWritePersistentData.START:= FALSE; 
						FB_WritePersistentDataDK_M_nEnable_iState:= 100;
					END_IF
				END_IF	
			END_IF

	006:	// Init
			M_nEnable:= cSTARTING;
			_fbWritePersistentData.START:= FALSE; 
			FB_WritePersistentDataDK_M_nEnable_iState:= FB_WritePersistentDataDK_M_nEnable_iState +1;

	007:	// Start
			M_nEnable:= cSTARTING;
			_fbWritePersistentData.START:= TRUE; 
			FB_WritePersistentDataDK_M_nEnable_iState:= FB_WritePersistentDataDK_M_nEnable_iState +1;
			
	008:	// Write persistent data - Done
			M_nEnable:= cSTARTING;
		
			// Error handling
			IF _fbWritePersistentData.ERR THEN
				M_nError(nErrorID:= _fbWritePersistentData.ERRID);	
				M_nEnable:= _fbWritePersistentData.ERRID;
			ELSE
				// Done
				IF NOT _fbWritePersistentData.BUSY THEN
					_nWriteCNT:= _nWriteCNT +1;
					_fbWritePersistentData.START:= FALSE; 
					FB_WritePersistentDataDK_M_nEnable_iState:= 100;
				END_IF	
			END_IF
	
	100:	// Done
			M_nEnable:= cCOMPLETE;
			_bFirstBoot:= FALSE;
			FB_WritePersistentDataDK_M_nEnable_iState:= 000;

ELSE
	FB_WritePersistentDataDK_M_nEnable_iState:= 000;	
END_CASE


// Proporty update
IF FB_WritePersistentDataDK_M_nEnable_fbStartDelay_TON.Q AND NOT _bPowerFailDetect AND NOT _bError THEN
	_bReady:= TRUE; 
ELSE
	_bReady:= FALSE; 
END_IF

// Status update
_fbWritePersistentData();
_bBusy:= _fbWritePersistentData.BUSY;
END_METHOD

//	The result of the method is an unsigned double integer
//	0 = idle 
//	1 = coupled
//	2 = starting
//	3 = running
//	4 = aborted
// 	5 = no hardware connected
//	7 = pointer or index error
//	8 = mapping error
//	9 = parameter error
//	10 = complete
//	Any other number = ErrorID
METHOD PUBLIC M_nWrite : UDINT
VAR_INPUT
	bExecute: BOOL;
END_VAR
//**********************************
// Reset 
//**********************************
IF _bReset THEN
	IF _bError THEN	
		FB_WritePersistentDataDK_M_nWrite_iState:= 000;
	END_IF	
END_IF

// Power fail
FB_WritePersistentDataDK_M_nWrite_fbReset_R_TRIG(CLK:= _bPowerFailDetect, Q=> );
IF FB_WritePersistentDataDK_M_nWrite_fbReset_R_TRIG.Q THEN
	FB_WritePersistentDataDK_M_nWrite_iState:= 000;
END_IF

//**********************************
// Wait for execute
//**********************************
IF FB_WritePersistentDataDK_M_nEnable_fbStartDelay_TON.Q THEN
	FB_WritePersistentDataDK_M_nWrite_fbExecute_R_TRIG(CLK:= bExecute AND NOT _bPowerFailDetect);
	IF FB_WritePersistentDataDK_M_nWrite_fbExecute_R_TRIG.Q THEN
		FB_WritePersistentDataDK_M_nWrite_iState:= 001;
	END_IF
ELSE
	FB_WritePersistentDataDK_M_nWrite_fbExecute_R_TRIG(CLK:= FALSE);
	FB_WritePersistentDataDK_M_nWrite_iState:= 000;
END_IF


//**********************************
// Main sekvens
//**********************************
CASE FB_WritePersistentDataDK_M_nWrite_iState OF

	000:	// Do nothing
	
	001:	// Running
			M_nWrite:= cRUNNING;
			IF _fbWritePersistentData.BUSY THEN
				FB_WritePersistentDataDK_M_nWrite_iState:= FB_WritePersistentDataDK_M_nWrite_iState +1;
			ELSE
				FB_WritePersistentDataDK_M_nWrite_iState:= FB_WritePersistentDataDK_M_nWrite_iState +2;
			END_IF

	002:	// Write persistent done
			M_nWrite:= cRUNNING;
			IF NOT _fbWritePersistentData.BUSY THEN
				_fbWritePersistentData.START:= FALSE; 
				FB_WritePersistentDataDK_M_nWrite_iState:= 100;
			END_IF
			
	003:	// Init
			M_nWrite:= cRUNNING;
			_fbWritePersistentData.START:= FALSE; 
			FB_WritePersistentDataDK_M_nWrite_iState:= FB_WritePersistentDataDK_M_nWrite_iState +1;

	004:	// Start
			M_nWrite:= cRUNNING;
			_fbWritePersistentData.START:= TRUE; 
			FB_WritePersistentDataDK_M_nWrite_iState:= FB_WritePersistentDataDK_M_nWrite_iState +1;

	005:	// Write persistent data - Done
			M_nWrite:= cRUNNING;
		
			// Error handling
			IF _fbWritePersistentData.ERR THEN
				M_nError(nErrorID:= _fbWritePersistentData.ERRID);	
				M_nWrite:= _fbWritePersistentData.ERRID;
			ELSE
				// Done
				IF NOT _fbWritePersistentData.BUSY THEN
					_nWriteCNT:= _nWriteCNT +1;
					_fbWritePersistentData.START:= FALSE; 	
					FB_WritePersistentDataDK_M_nWrite_iState:= 100;
				END_IF	
			END_IF
	
	100:	// Done
			M_nWrite:= cCOMPLETE;
			IF NOT bExecute THEN
				FB_WritePersistentDataDK_M_nWrite_iState:= 000;	
			END_IF	
	
ELSE
	FB_WritePersistentDataDK_M_nWrite_iState:= 000;	
END_CASE
END_METHOD

PROPERTY PUBLIC P_bBusy : BOOL
GET
P_bBusy:= _bBusy;
END_GET
END_PROPERTY

PROPERTY PUBLIC P_bPowerFailDetect : BOOL
GET
P_bPowerFailDetect:= _bPowerFailDetect;
END_GET
END_PROPERTY

PROPERTY PUBLIC P_eSUPS_Mode : Tc2_SUPS.E_S_UPS_Mode
SET
_eUpsMode:= P_eSUPS_Mode;
END_SET
END_PROPERTY

PROPERTY PUBLIC P_nWriteCNT : UDINT
GET
P_nWriteCNT:= _nWriteCNT;
END_GET
END_PROPERTY

END_FUNCTION_BLOCK
